FUNCTION_BLOCK FB_Transfo_Base
//////////////////
// High Voltage transformer with Transfo or DMCR detection . 
//////////////////

VAR_INPUT PERSISTENT
	// Parameters of the Object (instance/model specific) 
	ParamTimeOut_Alarm   		    : TIME  := T#200MS  ;		(* (ms) Config : Tempo when open and close before raising alarm*)

END_VAR

VAR_OUTPUT
	//Child objects
	
END_VAR

VAR_INPUT
		// Transfo

END_VAR

VAR
	///MesDataExd					: Transfo ; 
		MesCP_Read					: BOOL := TRUE;	(* Read function enable *)
		MesCP_Write					: BOOL := TRUE;	(* Write function enable *)	
END_VAR

METHOD M_AlarmManagement
//////////////////
// Manages High Voltage Transformer Alarms
/////////////////

VAR 
	// Method local variables (reinitialized at each cycle) 
	FB_AlarmCodeManager : FB_AlarmCodeManager ; 

	
END_VAR
END_METHOD

METHOD M_Execute
//////////////////
//  Method Calls 
/////////////////

VAR 
	// Method local variables (reinitialized at each cycle) 

END_VAR

	
// METHODS CALLS //
	M_Read();
	M_AlarmManagement();
END_METHOD

METHOD M_Read : BOOL
VAR_INPUT
END_VAR

VAR
	MesAuxTransfoGazDischarge: INT;
	MesAuxTransfoTempTrigger: INT;
END_VAR
END_METHOD

END_FUNCTION_BLOCK

(* stored: Version 1.1.0.1, ProductVersion 3.1.4024.12
   POU FB_Transfo_Base: Id {9b984ba0-2852-4da5-9ab0-fd011ae27334}, SpecialFunc None
   Method M_AlarmManagement: Id {d768a909-6eb6-4196-b98d-5eff50008abf}
   Method M_Execute: Id {f9ba8ac4-663e-4d75-abe1-1e0df67aa73b}
   Method M_Read: Id {b121c10b-dc3e-473f-8f52-1a7929ee3117} *)
